// Mitsubishi GX Works2 project: 12   PLC: FX3U/FX3UC

PROGRAM MAIN
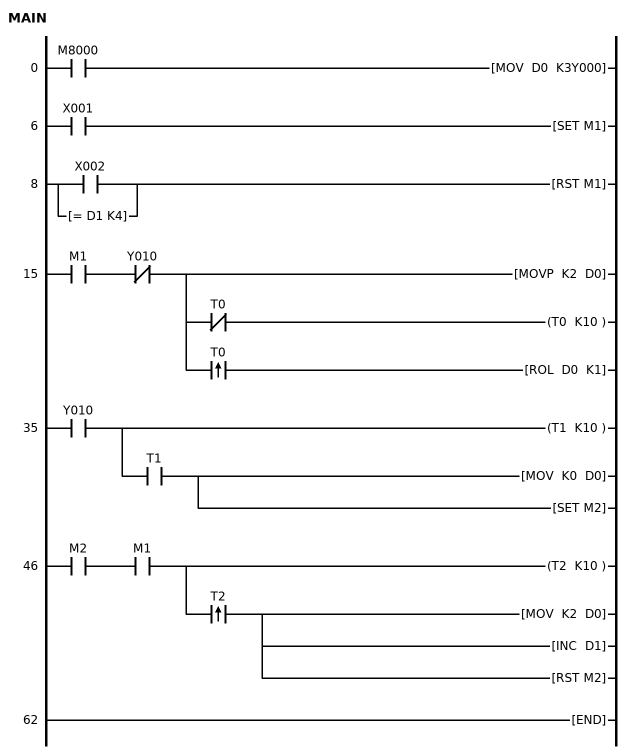
0     LD      M8000
      MOV     D0 K3Y000
6     LD      X001
      SET     M1
8     LD      X002
      OR=     D1 K4
      RST     M1
15    LD      M1
      ANI     Y010
      MOVP    K2 D0
      MPS
      ANI     T0
      OUT     T0 K10
      MPP
      ANDP    T0
      ROL     D0 K1
35    LD      Y010
      OUT     T1 K10
      AND     T1
      MOV     K0 D0
      SET     M2
46    LD      M2
      AND     M1
      OUT     T2 K10
      ANDP    T2
      MOV     K2 D0
      INC     D1
      RST     M2
62    END
END_PROGRAM
